// TwinCAT 3 PLC project PLC
// ProgramVersion: 3.1.4024.0
// libraries:
//   EfficientIO Communicator, * (EfficientIO)
//   EfficientIO Energy Basic, * (EfficientIO)
//   EfficientIO ModbusTCP, * (EfficientIO)
//   Lynus Energy ModbusRTU, * (Lynus AG)
//   Lynus Persistent Data V1, * (Lynus AG)
//   Lynus Standards, * (EfficientIO)
//   Tc2_Math, * (Beckhoff Automation GmbH)
//   Tc2_MBus, * (Beckhoff Automation GmbH)
//   Tc2_Standard, * (Beckhoff Automation GmbH)
//   Tc2_System, * (Beckhoff Automation GmbH)
//   Tc2_Utilities, * (Beckhoff Automation GmbH)
//   Tc3_JsonXml, * (Beckhoff Automation GmbH)
//   Tc3_Module, * (Beckhoff Automation GmbH)
// project tree:
//   / Fast_Task.TcTTO, Middle_Task.TcTTO, Slow_Task.TcTTO
//   FB/ FB_Delta_PV_Inverter_Sunspec.TcPOU (not stored), FB_KL6xxx_ModbusRTU_22B_Master.TcPOU, FB_Shelly_3EM.TcPOU (not stored), FB_Shelly_3EM_Helper.TcPOU (not stored), FB_Shelly_HT.TcPOU (not stored), FB_Shelly_HTplus.TcPOU (not stored), FB_Shelly_HTplus_Helper.TcPOU (not stored), FB_Shelly_HT_Helper.TcPOU
//   POUs/ MAIN.TcPOU, prgComEffIO.TcPOU (not stored), prgEM.TcPOU, prgEMS.TcPOU, prgGrid.TcPOU, prgHouse.TcPOU, prgMBUS.TcPOU, prgPersistent.TcPOU (not stored), prgPV.TcPOU, prgRWEffIO.TcPOU, prgVarEffIO.TcPOU (not stored)
// real-time tasks:
//   TASK Fast Task: cycle T#8ms, priority 8, ADS port 350
//   TASK Middle Task: cycle T#10ms, priority 10, ADS port 351
//   TASK Slow Task: cycle T#20ms, priority 20, ADS port 352
// I/O:
//   DEVICE Gerät 1 (Beckhoff CCAT)
//   DEVICE Gerät 2 (EtherCAT), AmsNetId 5.146.124.165.3.1
//     Klemme 1 (EK1200) [EK1200-5000 EtherCAT Netzteil (2A E-Bus)]
//       43A7_UV_Müller_Holzbau (EL3443-0010) [EL3443-0010 3K. Leistungsmessung 10A]
//       43A7.1_Abgang_Mieter (EL3443-0010) [EL3443-0010 3K. Leistungsmessung 10A]
//       43A8_Produktion_PV (EL3443-0010) [EL3443-0010 3K. Leistungsmessung 10A]
//       Klemme 5 (EL9010) [EL9010 Endklemme]
//   DEVICE Gerät 3 (RT-Ethernet Protocol), AmsNetId 5.146.124.165.4.1
//     BK9050 (BK9050-0000 192.168.1.118)
// variable links:
//   PLC/PLC Instance <-> Device 2 (EtherCAT)/Term 1 (EK1200)/43A7.1_Abgang_Mieter (EL3443-0010)
//     Middle_Task Inputs/prgHouse.ActivePowerTotal_2 <-> Total Active/Active Power
//   PLC/PLC Instance <-> Device 2 (EtherCAT)/Term 1 (EK1200)/43A7_UV_Müller_Holzbau (EL3443-0010)
//     Middle_Task Inputs/prgHouse.ActivePowerTotal_1 <-> Total Active/Active Power
//     Slow_Task Inputs/prgHouse.Strom1L1 <-> L1 Basic/Current
//     Slow_Task Inputs/prgHouse.Volt1L1 <-> L1 Basic/Voltage
//   PLC/PLC Instance <-> Device 2 (EtherCAT)/Term 1 (EK1200)/43A8_Produktion_PV (EL3443-0010)
//     Slow_Task Inputs/prgHouse.ActivePowerTotal_3 <-> Total Active/Active Power
//   PLC/PLC Instance <-> Device 3 (RT-Ethernet Protocol)/BK9050 (BK9050-0000 192.168.1.118)
//     Fast_Task Inputs/prgMBUS.stComIn @bit {16..184 step 8} <-> Term 2 (KL6781)/Channel 1/Data In {0..21}  (22 links)
//     Fast_Task Inputs/prgMBUS.stComIn <-> Term 2 (KL6781)/Channel 1/Status
//     Fast_Task Outputs/prgMBUS.stComOut <-> Term 2 (KL6781)/Channel 1/Ctrl
//     Fast_Task Outputs/prgMBUS.stComOut @bit {16..184 step 8} <-> Term 2 (KL6781)/Channel 1/Data Out {0..21}  (22 links)
//     Middle_Task Inputs/prgHouse.fbGrid1.fbKL3403.byStateCH1 <-> Elektromobilität (KL3403)/Channel 1/Status
//     Middle_Task Inputs/prgHouse.fbGrid1.fbKL3403.byStateCH2 <-> Elektromobilität (KL3403)/Channel 2/Status
//     Middle_Task Inputs/prgHouse.fbGrid1.fbKL3403.byStateCH3 <-> Elektromobilität (KL3403)/Channel 3/Status
//     Middle_Task Inputs/prgHouse.fbGrid1.fbKL3403.iDataInCH1 <-> Elektromobilität (KL3403)/Channel 1/Daten Ein
//     Middle_Task Inputs/prgHouse.fbGrid1.fbKL3403.iDataInCH2 <-> Elektromobilität (KL3403)/Channel 2/Daten Ein
//     Middle_Task Inputs/prgHouse.fbGrid1.fbKL3403.iDataInCH3 <-> Elektromobilität (KL3403)/Channel 3/Daten Ein
//     Middle_Task Inputs/prgHouse.fbGrid2.fbKL3403.byStateCH1 <-> Holzschnitzelheizung (KL3403)/Channel 1/Status
//     Middle_Task Inputs/prgHouse.fbGrid2.fbKL3403.byStateCH2 <-> Holzschnitzelheizung (KL3403)/Channel 2/Status
//     Middle_Task Inputs/prgHouse.fbGrid2.fbKL3403.byStateCH3 <-> Holzschnitzelheizung (KL3403)/Channel 3/Status
//     Middle_Task Inputs/prgHouse.fbGrid2.fbKL3403.iDataInCH1 <-> Holzschnitzelheizung (KL3403)/Channel 1/Daten Ein
//     Middle_Task Inputs/prgHouse.fbGrid2.fbKL3403.iDataInCH2 <-> Holzschnitzelheizung (KL3403)/Channel 2/Daten Ein
//     Middle_Task Inputs/prgHouse.fbGrid2.fbKL3403.iDataInCH3 <-> Holzschnitzelheizung (KL3403)/Channel 3/Daten Ein
//     Middle_Task Inputs/prgHouse.fbGrid3.fbKL3403.byStateCH1 <-> Lüftung_Kälte_Büro (KL3403)/Channel 1/Status
//     Middle_Task Inputs/prgHouse.fbGrid3.fbKL3403.byStateCH2 <-> Lüftung_Kälte_Büro (KL3403)/Channel 2/Status
//     Middle_Task Inputs/prgHouse.fbGrid3.fbKL3403.byStateCH3 <-> Lüftung_Kälte_Büro (KL3403)/Channel 3/Status
//     Middle_Task Inputs/prgHouse.fbGrid3.fbKL3403.iDataInCH1 <-> Lüftung_Kälte_Büro (KL3403)/Channel 1/Daten Ein
//     Middle_Task Inputs/prgHouse.fbGrid3.fbKL3403.iDataInCH2 <-> Lüftung_Kälte_Büro (KL3403)/Channel 2/Daten Ein
//     Middle_Task Inputs/prgHouse.fbGrid3.fbKL3403.iDataInCH3 <-> Lüftung_Kälte_Büro (KL3403)/Channel 3/Daten Ein
//     Middle_Task Outputs/prgHouse.fbGrid1.fbKL3403.byCntrCH1 <-> Elektromobilität (KL3403)/Channel 1/Kontrolle
//     Middle_Task Outputs/prgHouse.fbGrid1.fbKL3403.byCntrCH2 <-> Elektromobilität (KL3403)/Channel 2/Kontrolle
//     Middle_Task Outputs/prgHouse.fbGrid1.fbKL3403.byCntrCH3 <-> Elektromobilität (KL3403)/Channel 3/Kontrolle
//     Middle_Task Outputs/prgHouse.fbGrid2.fbKL3403.byCntrCH1 <-> Holzschnitzelheizung (KL3403)/Channel 1/Kontrolle
//     Middle_Task Outputs/prgHouse.fbGrid2.fbKL3403.byCntrCH2 <-> Holzschnitzelheizung (KL3403)/Channel 2/Kontrolle
//     Middle_Task Outputs/prgHouse.fbGrid2.fbKL3403.byCntrCH3 <-> Holzschnitzelheizung (KL3403)/Channel 3/Kontrolle
//     Middle_Task Outputs/prgHouse.fbGrid3.fbKL3403.byCntrCH1 <-> Lüftung_Kälte_Büro (KL3403)/Channel 1/Kontrolle
//     Middle_Task Outputs/prgHouse.fbGrid3.fbKL3403.byCntrCH2 <-> Lüftung_Kälte_Büro (KL3403)/Channel 2/Kontrolle
//     Middle_Task Outputs/prgHouse.fbGrid3.fbKL3403.byCntrCH3 <-> Lüftung_Kälte_Büro (KL3403)/Channel 3/Kontrolle

CONFIGURATION PLC
    RESOURCE PLC ON TwinCAT3
        TASK Fast_Task(INTERVAL := T#8ms, PRIORITY := 8);
        TASK Middle_Task(INTERVAL := T#10ms, PRIORITY := 10);
        TASK Slow_Task(INTERVAL := T#20ms, PRIORITY := 20);
        PROGRAM prgVarEffIO WITH Fast_Task : prgVarEffIO;
        PROGRAM prgRWEffIO WITH Fast_Task : prgRWEffIO;
        PROGRAM prgMBUS WITH Fast_Task : prgMBUS;
        PROGRAM prgPV WITH Fast_Task : prgPV;
        PROGRAM prgHouse WITH Middle_Task : prgHouse;
        PROGRAM prgGrid WITH Middle_Task : prgGrid;
        PROGRAM prgPersistent WITH Middle_Task : prgPersistent;
        PROGRAM prgEMS WITH Middle_Task : prgEMS;
        PROGRAM prgComEffIO WITH Slow_Task : prgComEffIO;
    END_RESOURCE
END_CONFIGURATION

// ---- POUs/prgRWEffIO.TcPOU
PROGRAM prgRWEffIO
VAR
	fbRW1		: FB_ReadWrite_V2;
END_VAR

fbRW1(
	eUploadType:= 3, // Change + 5 min Intervall 
	bBusy=> , 
	bError=> , 
	udiErrorCodeOut=> , 
	eErrorReadWrite_Out=> );

END_PROGRAM

// ---- POUs/prgMBUS.TcPOU
PROGRAM prgMBUS
VAR
	// M-Bus Kommunikation (KL6781)
	fbMBusKL6781         : FB_MBUSKL6781;             // Hauptbaustein für die M-Bus-Kommunikation
	stComIn              AT %I* : ST_KL6781inData22B; // Eingabestruktur für KL6781
	stComOut             AT %Q* : ST_KL6781outData22B;// Ausgabestruktur für KL6781
	stCom                : ST_MBUS_Communication;     // Kommunikationsstruktur für alle M-Bus-Geräte
	fbScann              : FB_MBUS_Scan;
	// Wärmezähler (Supercal 531)
	fbHolzkessel         : FB_MBUS_General;          	 // Funktionsbaustein für Holzkessel
	fbFussbodenheizung   : FB_MBUS_General;   		 	 // Funktionsbaustein für MAB Fußbodenheizung
	fbDSP_Produktion     : FB_MBUS_General;   			// Funktionsbaustein für DSP Produktion
	fbHeizkoerper_buero  : FB_MBUS_General;   			// Funktionsbaustein für Heizkörper Büro
	fbHalle_Bestand_S100 : FB_MBUS_General;   			// Funktionsbaustein für Halle Bestand S100
	fbLueftung	         : FB_MBUS_General;   			// Funktionsbaustein für Lüftung

	// Variablen für Steuerung
	m_Start1             : BOOL;                      
	m_Start2             : BOOL;                      
	m_Start3             : BOOL;
	m_Start4             : BOOL;
	m_Start5             : BOOL;
	m_Start6             : BOOL;
	
	//
	//TODO austausch FLOW mit Vorlauf und Rücklauftemperatur
	//
	
	// Ausgelesene Werte Wärmezähler
	lrEnergy_Holzkessel	 		: LREAL;								//{#lynus.ag#()}
	rFlow_Holzkessel     		: REAL;
	rPower_Holzkessel    		: REAL;									//{#lynus.ag#()}
	rflow_VL_Holzkessel			: REAL;									//{#lynus.ag#()}
	rflow_RL_Holzkessel			: REAL;									//{#lynus.ag#()}

	lrEnergy_Fussboden   		: LREAL;								//{#lynus.ag#()}
	rFlow_Fussboden         	: REAL;
	rPower_Fussboden        	: REAL;									//{#lynus.ag#()}
	rflow_VL_Fussboden			: REAL;									//{#lynus.ag#()}
	rflow_RL_Fussboden			: REAL;									//{#lynus.ag#()}

	lrEnergy_DSP_Produktion 	: LREAL;								//{#lynus.ag#()}
	rFlow_DSP_Produktion    	: REAL;
	rPower_DSP_Produktion   	: REAL;									//{#lynus.ag#()}
	rflow_VL_DSP_Produktion		: REAL;									//{#lynus.ag#()}
	rflow_RL_DSP_Produktion		: REAL;									//{#lynus.ag#()}
	
	lrEnergy_Heizkoerper_buero  : LREAL;								//{#lynus.ag#()}
	rFlow_Heizkoerper_buero     : REAL;
	rPower_Heizkoerper_buero    : REAL;									//{#lynus.ag#()}
	rflow_VL_Heizkoerper_buero	: REAL;									//{#lynus.ag#()}
	rflow_RL_Heizkoerper_buero	: REAL;									//{#lynus.ag#()}
	
	lrEnergy_Halle_Bestand_S100 : LREAL;								//{#lynus.ag#()}
	rFlow_Halle_Bestand_S100    : REAL;
	rPower_Halle_Bestand_S100   : REAL;									//{#lynus.ag#()}
	rflow_VL_Halle_Bestand_S100	: REAL;									//{#lynus.ag#()}
	rflow_RL_Halle_Bestand_S100	: REAL;									//{#lynus.ag#()}
	
	lrEnergy_Lueftung           : LREAL;								//{#lynus.ag#()}
	rFlow_Lueftung              : REAL;
	rPower_Lueftung             : REAL;									//{#lynus.ag#()}
	rflow_VL_Lueftung			: REAL;									//{#lynus.ag#()}
	rflow_RL_Lueftung			: REAL;									//{#lynus.ag#()}

	Err1 : E_MBUS_ERROR;
	Err2 : E_MBUS_ERROR;
	Err3 : E_MBUS_ERROR;
	Err4 : E_MBUS_ERROR;
	Err5 : E_MBUS_ERROR;
	Err6 : E_MBUS_ERROR;
	
	Busy1Trig : R_TRIG;
	DataReadyCount : DINT;
	DevError : ST_MBus_Info; 

	DataReadyCount2 : DINT;
	DevError2       : ST_MBus_Info; 

END_VAR

// ** M-Bus Hauptkommunikation **

fbMBusKL6781(
	usiRetries := 3,                    // Anzahl der Wiederholungen bei Fehler
	bStart := TRUE,                     // Startet die M-Bus-Kommunikation
	bDisabled := FALSE,                 // Deaktiviert die M-Bus-Kommunikation nicht
	bBusy => , 
	bReady => , 
	bError => , 
	eError => , 
	stComIn := stComIn, 
	stComOut := stComOut, 
	stCom := stCom
);

fbScann(
	bStart:= , 
	bStop:= , 
	eBaudrate:= E_MBUS_Baudrate.eMBus_Baud2400, 
	bDisabled:= , 
	bBusy=> , 
	bReady=> , 
	bError=> , 
	eError=> , 
	usiAddress=> , 
	usiCount=> , 
	arrDevice=> , 
	stCom:= stCom);


// ** Holzkessel (Supercal 531) auslesen **

//fbSupercal1.stSecAdr.udiIdNumber:= 30868639;

fbHolzkessel(
	usiAddress 	:= 1,                    	// M-Bus-Adresse(Primär)
	bStart 		:= m_Start1,                // Startflag
	usiUnit     := 1,               		// KW
	bDisabled 	:= FALSE,                 	
	bBusy => , 
	bReady => ,              				// Datenbereit-Status
	bError => , 
	eError => , 
	stCom 		:= stCom
);

IF NOT fbHolzkessel.bBusy AND fbHolzkessel.bError THEN

	Err1:= fbHolzkessel.eError;
END_IF

IF fbHolzkessel.bReady THEN

    lrEnergy_Holzkessel 	:= STRING_TO_REAL(fbHolzkessel.arrData[1].sValue);                 	// Energie (kWh)
    rFlow_Holzkessel 		:= STRING_TO_REAL(fbHolzkessel.arrData[6].sValue);                  // Durchfluss (m³/h)
    rPower_Holzkessel 	:= STRING_TO_REAL(fbHolzkessel.arrData[7].sValue);                    	// Leistung (kW)
END_IF

fbFussbodenheizung(
	usiAddress 	:= 2,                    	// M-Bus-Adresse(Primär)
	bStart 		:= m_Start2,                // Startflag
	usiUnit     := 1,               		// KW
	bDisabled 	:= FALSE,                 	
	bBusy => , 
	bReady => ,              				// Datenbereit-Status
	bError => , 
	eError => , 
	stCom 		:= stCom
);

IF NOT fbFussbodenheizung.bBusy AND fbFussbodenheizung.bError THEN

	Err2:= fbFussbodenheizung.eError;
END_IF

IF fbFussbodenheizung.bReady THEN

    lrEnergy_Fussboden 	:= STRING_TO_REAL(fbFussbodenheizung.arrData[1].sValue);                // Energie (kWh)
    rFlow_Fussboden 	:= STRING_TO_REAL(fbFussbodenheizung.arrData[6].sValue);                // Durchfluss (m³/h)
    rPower_Fussboden 	:= STRING_TO_REAL(fbFussbodenheizung.arrData[7].sValue);                // Leistung (kW)
	rflow_VL_Fussboden	:= STRING_TO_REAL(fbFussbodenheizung.arrData[3].sValue);					// Temperatur in Grad C
	rflow_RL_Fussboden	:= STRING_TO_REAL(fbFussbodenheizung.arrData[4].sValue);					// Temperatur in Grad C
END_IF

fbDSP_Produktion(
	usiAddress 	:= 3,                    	// M-Bus-Adresse(Primär)
	bStart 		:= m_Start3,                // Startflag
	usiUnit     := 1,               		// KW
	bDisabled 	:= FALSE,                 	
	bBusy => , 
	bReady => ,              				// Datenbereit-Status
	bError => , 
	eError => , 
	stCom 		:= stCom
);

IF NOT fbDSP_Produktion.bBusy AND fbDSP_Produktion.bError THEN

	Err3:= fbDSP_Produktion.eError;
END_IF

IF fbDSP_Produktion.bReady THEN

    lrEnergy_DSP_Produktion 	:= STRING_TO_REAL(fbDSP_Produktion.arrData[1].sValue);                 	// Energie (kWh)
    rFlow_DSP_Produktion 		:= STRING_TO_REAL(fbDSP_Produktion.arrData[6].sValue);                  // Durchfluss (m³/h)
    rPower_DSP_Produktion 		:= STRING_TO_REAL(fbDSP_Produktion.arrData[7].sValue);                  // Leistung (kW)
	rflow_VL_DSP_Produktion		:= STRING_TO_REAL(fbDSP_Produktion.arrData[3].sValue);					// Temperatur in Grad C
	rflow_RL_DSP_Produktion		:= STRING_TO_REAL(fbDSP_Produktion.arrData[4].sValue);					// Temperatur in Grad C
END_IF

fbHeizkoerper_buero(
	usiAddress 	:= 4,                    	// M-Bus-Adresse(Primär)
	bStart 		:= m_Start4,                // Startflag
	usiUnit     := 1,               		// KW
	bDisabled 	:= FALSE,                 	
	bBusy => , 
	bReady => ,              				// Datenbereit-Status
	bError => , 
	eError => , 
	stCom 		:= stCom
);

IF NOT fbHeizkoerper_buero.bBusy AND fbHeizkoerper_buero.bError THEN

	Err4:= fbHeizkoerper_buero.eError;
END_IF

IF fbHeizkoerper_buero.bReady THEN

    lrEnergy_Heizkoerper_buero 	:= STRING_TO_REAL(fbHeizkoerper_buero.arrData[1].sValue);                 	// Energie (kWh)
    rFlow_Heizkoerper_buero 	:= STRING_TO_REAL(fbHeizkoerper_buero.arrData[6].sValue);                  // Durchfluss (m³/h)
    rPower_Heizkoerper_buero 	:= STRING_TO_REAL(fbHeizkoerper_buero.arrData[7].sValue);                  // Leistung (kW)
	rflow_VL_Heizkoerper_buero	:= STRING_TO_REAL(fbHeizkoerper_buero.arrData[3].sValue);					// Temperatur in Grad C
	rflow_RL_Heizkoerper_buero	:= STRING_TO_REAL(fbHeizkoerper_buero.arrData[4].sValue);					// Temperatur in Grad C
END_IF

fbHalle_Bestand_S100(
	usiAddress 	:= 5,                    	// M-Bus-Adresse(Primär)
	bStart 		:= m_Start5,                // Startflag
	usiUnit     := 1,               		// KW
	bDisabled 	:= FALSE,                 	
	bBusy => , 
	bReady => ,              				// Datenbereit-Status
	bError => , 
	eError => , 
	stCom 		:= stCom
);

IF NOT fbHalle_Bestand_S100.bBusy AND fbHalle_Bestand_S100.bError THEN

	Err5:= fbHalle_Bestand_S100.eError;
END_IF

IF fbHalle_Bestand_S100.bReady THEN

    lrEnergy_Halle_Bestand_S100 	:= STRING_TO_REAL(fbHalle_Bestand_S100.arrData[1].sValue);                 	// Energie (kWh)
    rFlow_Halle_Bestand_S100 		:= STRING_TO_REAL(fbHalle_Bestand_S100.arrData[6].sValue);                  // Durchfluss (m³/h)
    rPower_Halle_Bestand_S100 		:= STRING_TO_REAL(fbHalle_Bestand_S100.arrData[7].sValue);                  // Leistung (kW)
	rflow_VL_Halle_Bestand_S100		:= STRING_TO_REAL(fbHalle_Bestand_S100.arrData[3].sValue);					// Temperatur in Grad C
	rflow_RL_Halle_Bestand_S100		:= STRING_TO_REAL(fbHalle_Bestand_S100.arrData[4].sValue);					// Temperatur in Grad C
END_IF


fbLueftung(
	usiAddress 	:= 6,                    	// M-Bus-Adresse(Primär)
	bStart 		:= m_Start6,                // Startflag
	usiUnit     := 1,               		// KW
	bDisabled 	:= FALSE,                 	
	bBusy => , 
	bReady => ,              				// Datenbereit-Status
	bError => , 
	eError => , 
	stCom 		:= stCom
);

IF NOT fbLueftung.bBusy AND fbLueftung.bError THEN

	Err6:= fbLueftung.eError;
END_IF

IF fbLueftung.bReady THEN

    lrEnergy_Lueftung 	:= STRING_TO_REAL(fbLueftung.arrData[1].sValue);             	// Energie (kWh)
    rFlow_Lueftung 		:= STRING_TO_REAL(fbLueftung.arrData[6].sValue);             	// Durchfluss (m³/h)
    rPower_Lueftung 	:= STRING_TO_REAL(fbLueftung.arrData[7].sValue);            	// Leistung (kW)
	rflow_VL_Lueftung	:= STRING_TO_REAL(fbLueftung.arrData[3].sValue);				// Temperatur in Grad C
	rflow_RL_Lueftung	:= STRING_TO_REAL(fbLueftung.arrData[4].sValue);				// Temperatur in Grad C
END_IF

END_PROGRAM

// ---- POUs/prgPV.TcPOU
PROGRAM prgPV
VAR
	//fbPV1							:FB_SunSpec_PV_Inverter;
	Wechselrichter1kWRaw AT %MW0	:INT;
	Wechselrichter1kW				:REAL;							//{#lynus.ag#()}
	Wechselrichter2kWRaw AT %MW2	:INT;
	Wechselrichter2kW				:REAL;							//{#lynus.ag#()}
	Wechselrichter3kWRaw AT %MW4	:INT;
	Wechselrichter3kW				:REAL;							//{#lynus.ag#()}
	Wechselrichter4kWRaw AT %MW6	:INT;
	Wechselrichter4kW				:REAL;							//{#lynus.ag#()}
	Wechselrichter5kWRaw AT %MW8	:INT;
	Wechselrichter5kW				:REAL;							//{#lynus.ag#()}
	Wechselrichter6kWRaw AT %MW10	:INT;
	Wechselrichter6kW				:REAL;							//{#lynus.ag#()}
	Wechselrichter7kWRaw AT %MW12	:INT;
	Wechselrichter7kW				:REAL;							//{#lynus.ag#()}
	Wechselrichter8kWRaw AT %MW14	:INT;
	Wechselrichter8kW				:REAL;							//{#lynus.ag#()}
	Wechselrichter9kWRaw AT %MW16	:INT;
	Wechselrichter9kW				:REAL;							//{#lynus.ag#()}
	PV_Gesamt						:REAL;							//{#lynus.ag#()}

END_VAR

Wechselrichter1kW := TO_REAL(Wechselrichter1kWRaw) / 100.0;
Wechselrichter2kW := TO_REAL(Wechselrichter2kWRaw) / 100.0;
Wechselrichter3kW := TO_REAL(Wechselrichter3kWRaw) / 100.0;
Wechselrichter4kW := TO_REAL(Wechselrichter4kWRaw) / 100.0;
Wechselrichter5kW := TO_REAL(Wechselrichter5kWRaw) / 100.0;
Wechselrichter6kW := TO_REAL(Wechselrichter6kWRaw) / 100.0;
Wechselrichter7kW := TO_REAL(Wechselrichter7kWRaw) / 100.0;
Wechselrichter8kW := TO_REAL(Wechselrichter8kWRaw) / 100.0;
Wechselrichter9kW := TO_REAL(Wechselrichter9kWRaw) / 100.0;

PV_Gesamt 		  := Wechselrichter1kW + Wechselrichter2kW + Wechselrichter3kW + Wechselrichter4kW + Wechselrichter5kW + Wechselrichter6kW + Wechselrichter7kW + Wechselrichter8kW + Wechselrichter9kW;

(*
fbPV1(
	bEnable:= , 
	sIPAdress:= '192.168.140.6', 
	byUnitID_Inverter:= 1, 
	stDataSunSpec=> , 
	stDataEMPower_PV=> , 
	stDataEMCounter_PV=> , 
	diNrOfEM_OUT_PV=> 
);
*)

END_PROGRAM

// ---- POUs/prgHouse.TcPOU
PROGRAM prgHouse
VAR
	fbKBusState					: FB_K_Bus_State;
	uint_KBusState				: UINT;							//{#lynus.ag#()}
	lrHousePower				: LREAL;								//{#lynus.ag#()}
	lrNetzEinspeisung			: LREAL;								//{#lynus.ag#()}
	lrBetriebMuellerBau			: LREAL;								//{#lynus.ag#()}
	lrElektromobilitaet			: LREAL;								//{#lynus.ag#()}
	lrHolzschnitzel				: LREAL;								//{#lynus.ag#()}
	lrLueftung_Kaelte			: LREAL;								//{#lynus.ag#()}
	//rPVProd						: REAL;									//{#lynus.ag#()}
	lrAbgaenge					: REAL;									//{#lynus.ag#()}
	fbGrid1						: FB_EM_Beckhoff_KL3403;  	//Elektromobilität 
	fbGrid2						: FB_EM_Beckhoff_KL3403;	//Holzschnitzelheizung
	fbGrid3						: FB_EM_Beckhoff_KL3403;	//Lüftung/Kälte Büro
	
	

    Volt1L1  AT %I* : REAL;
    Strom1L1 AT %I* : REAL;
	//UV Müller Holzbau
	ActivePowerTotal_1	AT %I*	: REAL;									//{#lynus.ag#()}
	//Abgang Direktmessung
	ActivePowerTotal_2	AT %I*	: REAL;									//{#lynus.ag#()}
	//Produktion PV
	ActivePowerTotal_3	AT %I*	: REAL;									//{#lynus.ag#()}

END_VAR

lrNetzEinspeisung := ActivePowerTotal_1/1000 + ActivePowerTotal_2/1000 - prgPV.PV_Gesamt;

lrElektromobilitaet	:= fbGrid1.stDataEMPower.lrPowerTotal;
lrHolzschnitzel		:= fbGrid2.stDataEMPower.lrPowerTotal;
lrLueftung_Kaelte	:= fbGrid3.stDataEMPower.lrPowerTotal;
lrHousePower		:= ActivePowerTotal_1/1000 + fbGrid1.stDataEMPower.lrPowerTotal + fbGrid2.stDataEMPower.lrPowerTotal + fbGrid3.stDataEMPower.lrPowerTotal;

lrBetriebMuellerBau := -fbGrid1.stDataEMPower.lrPowerTotal - fbGrid2.stDataEMPower.lrPowerTotal - fbGrid3.stDataEMPower.lrPowerTotal + lrHousePower;	

//rPVProd				:= (ActivePowerTotal_3)/100 * -1;					//Invertieren
lrAbgaenge 			:= ActivePowerTotal_2/1000;
//lrHousePower 		:= lrBetriebMuellerBau * -1;						//Invertierte Einspeisung für Darstellung

//The mapping of this function must be linked with the K-Bus State in the E/A Part
fbKBusState(	uiKBusState_OUT=> , 
				b_Kbus_notOk=> , 
				word_ErrorCount=> );

fbGrid1(
	bEnable:= TRUE, 
	bChannel1Invers:= FALSE, 
	bChannel2Invers:= FALSE, 
	bChannel3Invers:= FALSE, 
	uiCurrentTransformerRatioL1:= 400, 
	uiCurrentTransformerRatioL2:= 400, 
	uiCurrentTransformerRatioL3:= 400, 
	uiKBusState_IN:= fbKBusState.uiKBusState_OUT, 
	stDataEMPower=> , 
	stDataEMCounter=> , 
	stDataEMPowerRealTime=> , 
	stDataEMCounterRealTime=> , 
	diNrOfEM_OUT=> );
	
	
fbGrid2(
	bEnable:= TRUE, 
	bChannel1Invers:= FALSE, 
	bChannel2Invers:= FALSE, 
	bChannel3Invers:= FALSE, 
	uiCurrentTransformerRatioL1:= 400, 
	uiCurrentTransformerRatioL2:= 400, 
	uiCurrentTransformerRatioL3:= 400, 
	uiKBusState_IN:= , 
	stDataEMPower=> , 
	stDataEMCounter=> , 
	stDataEMPowerRealTime=> , 
	stDataEMCounterRealTime=> , 
	diNrOfEM_OUT=> );
	
fbGrid3(
	bEnable:= TRUE, 
	bChannel1Invers:= FALSE, 
	bChannel2Invers:= FALSE, 
	bChannel3Invers:= FALSE, 
	uiCurrentTransformerRatioL1:= 400, 
	uiCurrentTransformerRatioL2:= 400, 
	uiCurrentTransformerRatioL3:= 400, 
	uiKBusState_IN:= , 
	stDataEMPower=> , 
	stDataEMCounter=> , 
	stDataEMPowerRealTime=> , 
	stDataEMCounterRealTime=> , 
	diNrOfEM_OUT=> );

END_PROGRAM

// ---- POUs/prgGrid.TcPOU
PROGRAM prgGrid
VAR
	fbKBusState					: FB_K_Bus_State;
	fbGrid						: FB_EM_Beckhoff_KL3403;
	uint_KBusState				: UINT;							//{#lynus.ag#()}
	fbGridCounter				: FB_EnergyCounter;
	lrGridPower					: LREAL;								//{#lynus.ag#()}
	lrVoltage_L1N					: LREAL;								//{#lynus.ag#()}
	lrVoltage_L2N					: LREAL;								//{#lynus.ag#()}
	lrVoltage_L3N					: LREAL;								//{#lynus.ag#()}
END_VAR
VAR PERSISTENT
	rSizeGridConn				: REAL;									//{#lynus.ag#()}
	lrCounterGridProd			: LREAL;								//{#lynus.ag#()}
	lrCounterGridCons			: LREAL;								//{#lynus.ag#()}
END_VAR

//The mapping of this function must be linked with the K-Bus State in the E/A Part
fbKBusState(	uiKBusState_OUT=> , 
				b_Kbus_notOk=> , 
				word_ErrorCount=> );

//The mapping of this function must be linked with the KL3403 in the E/A Part
//UV1
fbGrid(
	bEnable:= TRUE, 
	bChannel1Invers:= FALSE,				//Invert power data when transformer are mounted upside down
	bChannel2Invers:= FALSE,			// CT seems to be wired the wrong wy around
	bChannel3Invers:= FALSE,
	uiCurrentTransformerRatioL1:= 400, //Transformer ratio on the secondary side
	uiCurrentTransformerRatioL2:= 400, 
	uiCurrentTransformerRatioL3:= 400, 
	uiKBusState_IN:= fbKBusState.uiKBusState_OUT, 
	stDataEMPower=> , 
	stDataEMCounter=> , 
	stDataEMPowerRealTime=> , 
	stDataEMCounterRealTime=> , 
	diNrOfEM_OUT=> );
	
uint_KBusState :=	fbKBusState.uiKBusState_OUT;
lrGridPower := fbGrid.stDataEMPower.lrPowerTotal;

// EnergyCounter
fbGridCounter(
	byActiveTariff:= 1, 
	lrPowerInput:= lrGridPower, 
	lrTotalCounterEnergy_Consumption=> , 
	lrTotalCounterEnergy_Production=> , 
	lrCounterEnergyT1_Consumption=> , 
	lrCounterEnergyT2_Consumption=> , 
	lrCounterEnergyT1_Production=> , 
	lrCounterEnergyT2_Production=> );

IF fbGridCounter.lrTotalCounterEnergy_Production > lrCounterGridProd THEN  	
		lrCounterGridProd := fbGridCounter.lrTotalCounterEnergy_Production;
END_IF

IF fbGridCounter.lrTotalCounterEnergy_Consumption > lrCounterGridCons THEN  	
	lrCounterGridCons := fbGridCounter.lrTotalCounterEnergy_Consumption;
END_IF

lrVoltage_L1N := fbGrid.stDataEMPower.lrVoltageL1N;
lrVoltage_L2N := fbGrid.stDataEMPower.lrVoltageL2N;
lrVoltage_L3N := fbGrid.stDataEMPower.lrVoltageL3N;

END_PROGRAM

// ---- POUs/prgEMS.TcPOU
PROGRAM prgEMS
VAR PERSISTENT
	byMaxDepthOfDischrgEPO		: BYTE;							//{#lynus.ag#()}
	byPrioMinChrgBattSOCInEPO	: BYTE;							//{#lynus.ag#()}
	byResChrgfromGridToBatt		: BYTE;							//{#lynus.ag#()}
	byReserveSOCEPO				: BYTE;							//{#lynus.ag#()}
	uiUpdateTime				: UINT;							//{#lynus.ag#()}
	bEnableEMS					: BOOL;							//{#lynus.ag#()}
	bAllowChrgFromGrid			: BOOL;							//{#lynus.ag#()}
	rMainFuseCSEMS				: REAL;							//{#lynus.ag#()}
	iOperationModeEMS			: INT;							//{#lynus.ag#()}
	rSizeGridConn				: REAL;							//{#lynus.ag#()}
END_VAR
VAR
	fbEMS						: FB_EMS_V2;
	bIsEnableEMS				: BOOL;							//{#lynus.ag#()}
	bStateAllowChrgFromGrid		: BOOL;							//{#lynus.ag#()}
	bStateFuseCS				: BOOL;							//{#lynus.ag#()}
	bHPActivate					: BOOL;							//{#lynus.ag#()}
	bControllingState			: BOOL;							//{#lynus.ag#()}
	iMessageEMS					: INT;							//{#lynus.ag#()}
	rHeartbeatEMS				: REAL;							//{#lynus.ag#()}
	rErrorWarningEMS			: REAL;							//{#lynus.ag#()}
	rReadyEMS					: REAL;							//{#lynus.ag#()}
	rNewBatteryPowerEMS			: REAL;							//{#lynus.ag#()}
	fbGrid: FB_Grid_Power_Ext_Input;

END_VAR

IF iOperationModeEMS = 0 THEN fbEMS.eOperationMode := E_OperatingMode_EMS.eAllOff;
ELSIF iOperationModeEMS = 1 THEN fbEMS.eOperationMode := E_OperatingMode_EMS.eSelfConsumption;	
ELSIF iOperationModeEMS = 2 THEN fbEMS.eOperationMode := E_OperatingMode_EMS.ePeakLoadCapping;
ELSIF iOperationModeEMS = 3 THEN fbEMS.eOperationMode := E_OperatingMode_EMS.eLoadManagement;			
END_IF
fbEMS.stSetupEMS.bAllowChrgFromGrid := bAllowChrgFromGrid;
fbEMS.stSetupEMS.byMaxDepthOfDischrgEPO := byMaxDepthOfDischrgEPO;
// fbEMS.stSetupEMS.byPrioMinChrgBattSOCInEPO := byPrioMinChrgBattSOCInEPO;
// fbEMS.stSetupEMS.byResChrgfromGridToBatt := byResChrgfromGridToBatt;
fbEMS.stSetupEMS.byReserveSOCEPO := byReserveSOCEPO;
//fbEMS.stSetupEMS.rSizeMainFuseCS := rMainFuseCSEMS;
fbEMS.stSizeMainFuseCS.rElSizeLine1 := rMainFuseCSEMS;
fbEMS.stSetupEMS.bEnableMainFuseFunc := bStateFuseCS;
fbEMS.stSetupEMS.uiUpdateTime := uiUpdateTime;

fbEMS(
	bEnable						:= bEnableEMS, 
//	diNrOfEM_IN_ECS				:= , 
	stSetupEMS					:= , 
	eOperationMode				:= , 
	eSpeedModeBackendController	:= E_SpeedModeBackendController_EMS.eFast, 
	eSpeedModeLocalController	:= E_SpeedModeLocalController_EMS.eFast,
	bActivateHP					:= bHPActivate, 
	bControllingState			:= bControllingState, 
	rHeartbeat					:= rHeartbeatEMS, 
	rErrorWarning				:= rErrorWarningEMS, 
	rEnergyOptReady				:= rReadyEMS, 
	rNewBattPower				:= rNewBatteryPowerEMS, 

	eMessageEMS				=> iMessageEMS, 
	bStateEnable			=> bIsEnableEMS, 
	bStateAllowChrgFromGrid	=> bStateAllowChrgFromGrid, 
	bMissingPowerData		=> , 
	bSurplusAvailable		=> , 
	byProgress				=> , 
	uiState_OUT				=> , 
	diNrOfEMS_OUT			=> , 
	arrMinPrioReached		=> , 
	arrMaxPrioReached		=> ,
	);
	
fbGrid(
	bEnable:= TRUE, 
	diNrOfEMS_IN:= prgEMS.fbEMS.diNrOfEMS_OUT, 
	rSizeGridConn:= rSizeGridConn , 
	bExtErrorGrid:= , 
	lrExtGridPower:= prgHouse.lrNetzEinspeisung , 
	lrExtTotalCounterEnergy_Consumption:= , 
	lrExtTotalCounterEnergy_Production:= , 
	lrExtCounterEnergyT1_Consumption:= , 
	lrExtCounterEnergyT2_Consumption:= , 
	lrExtCounterEnergyT1_Production:= , 
	lrExtCounterEnergyT2_Production:= , 
	stDataGrid=> , 
	diNrOfGrid_OUT=> );

END_PROGRAM

// ---- FB/FB_KL6xxx_ModbusRTU_22B_Master.TcPOU
FUNCTION_BLOCK FB_KL6xxx_ModbusRTU_22B_Master
VAR_INPUT
	bConfigTerminal							: BOOL;																		//Possibility to configure the Terminal manually (Its only possible when the Terminal is not configured successfully)
	uiKBusState_IN							: UINT;																		//K-Bus State from the K-Bus Box on wich the Terminal is connected. (Connect with FB_K_Bus_state)
END_VAR
VAR_OUTPUT
	bBusy									: BOOL;																		//Function is Busy
	byErrorWarning							: BYTE;																		//Error Warning State
	byActualAdressInUse						: BYTE;																		//Actual Modbus Adress in Use
	diNrOfMBRTUMasterLine_OUT				: DINT;																		//Active Number from the RTU Master Function for using on other functions
	eMessageMBRTUMaster						: E_Message_MBRTUMaster;													//Message from the RTU Master Function
END_VAR				
VAR_OUTPUT PERSISTENT
	bTerminalIsConfigured					: BOOL;																		//Its True when the configuration is successfully
END_VAR
VAR		
	config_execute							: BOOL ;
	//{attribute 'hide'}
	fbKL6xxxConfig							: KL6configuration;															//FB KL6xxx to config the terminal
	fbmodbusmaster							: ModbusRtuMaster_KL6x22B;													//FB Modbus RTU
	{attribute 'hide'}
	fbmodbusmaster_Init						: ModbusRtuMaster_KL6x22B;													//FB Modbus RTU Master for workaroud regarding the internal Beckhoff problem in this function
	{attribute 'hide'}
	fbNumberDevice							: FB_NumberOfDevice;														//Function block to calcualte the number of the Device	
	{attribute 'hide'}
	fbModbusRTUMessage						: FB_MBRTUMaster_Messages;													//Modbus RTU Messages	
	{attribute 'hide'}
	FPConfigManual							: R_TRIG;																	//Internal positive Edge
	{attribute 'hide'}
	FPConfigAuto							: R_TRIG;																	//Internal positive Edge
	{attribute 'hide'}
	FPProcessCompleted						: R_TRIG;																	//Internal positive Edge
	{attribute 'hide'}
	FPError									: R_TRIG;																	//Internal positive Edge
	{attribute 'hide'}
	FPErrorIsActive							: R_TRIG;																	//Internal positive Edge
	{attribute 'hide'}
	FNInitSmall								: F_TRIG;																	//Internal negative Edge
	{attribute 'hide'}
	FNBusy									: F_TRIG;																	//Internal negative Edge
	{attribute 'hide'}
	timInit									: TON;																		//Delay to start the Terminal Configuration after the start from the plc
	{attribute 'hide'}
	timTimout								: TON;																		//Timer Timout to go on next Modbus Adress when the Ack is not set back to False
	{attribute 'hide'}
	timDissableFunctions					: TON;																		//Timer to dissable the Function after Lynus_Standards.Constants_General.tTimeDissableLynusFunctions Days without connection to the Lynus Cloud
	{attribute 'hide'}
	timResetConnectionOnGVL					: TON;																		//Timer to try reset the connection Flag on the GVL. (When somebody delete the Connection Function and make only a onlinechange)
	{attribute 'hide'}
	arrPD									: ARRAY[1..2] OF FB_PersistentData_Number;									//Function to save persistent data
	{attribute 'hide'}
	bTakeActualAdress						: BOOL;																		//True if the Current address is to be used
	{attribute 'hide'}
	bAdressHasChanged						: BOOL;																		//True if the Adress has changed
	{attribute 'hide'}
	bErrorIsActive							: BOOL;																		//True if a Error is happend. False after the next successfully read or write command
	{attribute 'hide'}
	bStopReadWrite							: BOOL;																		//Stop Function because Modbus Adress has chaged
	{attribute 'hide'}
	byLPSmallestAdress						: BYTE;																		//Loop to find out the smallest Modbus Adress
	{attribute 'hide'}
	byLPBiggestAdress						: BYTE;																		//Loop to find out the biggest Modbus Adress
	{attribute 'hide'}
	byLPActualAdress						: BYTE;																		//Loop to find out the next actuall adress
	{attribute 'hide'}
	byLPNumbersOfTotalSlaves				: BYTE;																		//Loop to find out the number of total Modbus Slaves
	{attribute 'hide'}
	bySmallestAdress						: BYTE;																		//Smallest Modbus Adress
	{attribute 'hide'}
	byBiggestAdress							: BYTE;																		//Biggest Modbus Adress
	{attribute 'hide'}
	byActualAdressInUse_CP					: BYTE;																		//Actual Modbus Adress in Use to compare it with the old one
	{attribute 'hide'}
	byNumberOfTotalSlaves					: BYTE;																		//Number of all Modbus Slaves
	{attribute 'hide'}
	byWaitInStep							: BYTE;																		//Wait in Step before start to clean data on PLC
	{attribute 'hide'}
	byLPMBAdress							: BYTE;																		//Loop for manage new Modbus Adress List after a change
	{attribute 'hide'}
	bySearchMBAdress						: BYTE;																		//Search Modbus Adress after change
	{attribute 'hide'}
	byPosInArrayMBAdress					: BYTE;																		//Save new Range from Modbus adress in the Array after a change
	{attribute 'hide'}
	iStateGVLData							: INT;																		//State machine to handle the data on the GVL
	{attribute 'hide'}
	iStateSetMBAdress						: INT;																		//State machin eto order the Modbus Adress after a change
	{attribute 'hide'}
	diCounterForGVL							: DINT;																		//Counter to clean old data on GVL
	{attribute 'hide'}
	arrRead									: ARRAY[1..Constants_Bussystems.wQuantityOfRegistersMBRTUMaster] OF WORD;	//Puffer for read out data
	{attribute 'hide'}
	arrMBAdress								: ARRAY[1..247] OF BYTE;													//Array with the actual Modbus Adress Config
END_VAR
VAR PERSISTENT
	{attribute 'conditionalshow'}
	eDeviceType								: E_MBRTUMaster_DeviceType;													//Device Type on witch the Terminal is configured
END_VAR

//Creator : Kai Ebensperger
//Company : Lynus AG
//Date : 08.07.2021
//Version : 1.0.0.0

//With this FB a serial 22 byte terminal can be configured and data can be sent/received via Modbus RTU.
//Only devices of the same type may be operated on the same master (because its not good to write to much new configurations on the terminal).
//The 1 slave that is called before the master FB in the PLC code configures the terminal
//The block must be called in a task of 5MS
//The system works according to the Master Slave principle
//Multiple communication is not possible in RTU principle

//NOTE for diNr.....Designation => 
//_IN = Here Data come in from other Functions or go out to other functions about the GVL
//_OUT = Here Data go out to other functions about the GVL

(*-------------------------------------------------------------Calcualte the number of RTU Master---------------------------------------------------------------*)

fbNumberDevice(
	diActualNumberOfDevices:= Lynus_Standards.GVL_Bussystems.diNumberOfMBRTUMasters, 
	diMaxNumberOfDevices:= Constants_Bussystems.diMaxNumberOfMBRTUMasterKL6xxx, 
	udiCounterOnlineChange:= TwinCAT_SystemInfoVarList._AppInfo.OnlineChangeCnt, 
	bNumberIsCalculatet=> , 
	bFPNumberIsCalculatet=> , 
	bOnlineChange=> , 
	diNumberForThisDevice=> diNrOfMBRTUMasterLine_OUT, 
	diNumberOfTotalDevices=> );

//Write new Numer on GVL
IF fbNumberDevice.bFPNumberIsCalculatet THEN
	Lynus_Standards.GVL_Bussystems.diNumberOfMBRTUMasters := fbNumberDevice.diNumberOfTotalDevices;	
END_IF 

//Delete old Number on GVL
IF fbNumberDevice.bOnlineChange THEN 
	Lynus_Standards.GVL_Bussystems.diNumberOfMBRTUMasters := diNrOfMBRTUMasterLine_OUT;	
		iStateGVLData := 1; 
END_IF	
	
(*-------------------------------------------------------------Service from Backend is ready and check the connection to backen for dissabel/enable Function---------------------------------------------------------------*)

//Try to reset the variable for connection on the GVL. When all is normal then the Lynus Mqtt connection function set this variable to true in the next cycle
//When we have no connection to the backend then after Lynus_Standards.Constants_General.tTimeDissableLynusFunctions days the Function is dissabled with all of his functionalities
timResetConnectionOnGVL(IN:= NOT timResetConnectionOnGVL.Q, PT:= T#1H, Q=> , ET=> );
	IF timResetConnectionOnGVL.Q THEN Lynus_Standards.GVL_Communicator.bStateConnectionToEnableFunctions := FALSE; END_IF
		IF NOT Lynus_Standards.GVL_Communicator.bStateConnectionToEnableFunctions THEN timDissableFunctions.IN := TRUE; ELSE timDissableFunctions.IN := FALSE; END_IF  
			timDissableFunctions(IN:= , PT:= Lynus_Standards.Constants_General.tTimeDissableLynusFunctions, Q=> , ET=> );

(*------------------------------------------------------------------Configuration----------------------------------------------------------------------------*)
			
//Configurate the seriall Terminal
//The configuration is depending what Slave is connected to the terminal
timInit(IN:= Lynus_Standards.GVL_Bussystems.stDataOfMBRTUMasterKL6xxx[diNrOfMBRTUMasterLine_OUT].eMBRTUDeviceType <> E_MBRTUMaster_DeviceType.eNoModbusRTUDevice AND uiKBusState_IN = 0, PT:=T#500MS, Q=> , ET=> );

IF Lynus_Standards.GVL_Bussystems.stDataOfMBRTUMasterKL6xxx[diNrOfMBRTUMasterLine_OUT].eMBRTUDeviceType <> eDeviceType AND timInit.Q THEN
	FPConfigAuto.CLK := TRUE;
		eDeviceType := Lynus_Standards.GVL_Bussystems.stDataOfMBRTUMasterKL6xxx[diNrOfMBRTUMasterLine_OUT].eMBRTUDeviceType;
ELSE
	FPConfigAuto.CLK := FALSE;
END_IF 	 

FPConfigAuto(CLK:= , Q=> );

//Configuration from the Terminal by the Slave Type
IF Lynus_Standards.GVL_Bussystems.stDataOfMBRTUMasterKL6xxx[diNrOfMBRTUMasterLine_OUT].eMBRTUDeviceType = E_MBRTUMaster_DeviceType.ePilotPMAC201_HW THEN
	//Pilot PMAC201 HW Energymessurement Device
	fbKL6xxxConfig.Mode := SERIALLINEMODE_KL6_22B_STANDARD;
	fbKL6xxxConfig.Baudrate := 38400;
	fbKL6xxxConfig.NoDatabits := 8;
	fbKL6xxxConfig.Parity := PARITY_NONE;
	fbKL6xxxConfig.Stopbits := 1;
	fbKL6xxxConfig.Handshake := RS485_HALFDUPLEX;
	fbKL6xxxConfig.ContinousMode := FALSE;
	//Timout	
	timTimout.PT := T#2S;
	fbmodbusmaster.Timeout := T#2S;
ELSIF Lynus_Standards.GVL_Bussystems.stDataOfMBRTUMasterKL6xxx[diNrOfMBRTUMasterLine_OUT].eMBRTUDeviceType = E_MBRTUMaster_DeviceType.eDrexelAWeiss_AereosilentStratosLU_Ventilation THEN
	//Aereosilent Stratos Ventilation Drexel and Weiss
	fbKL6xxxConfig.Mode := SERIALLINEMODE_KL6_22B_STANDARD;
	fbKL6xxxConfig.Baudrate := 19200;
	fbKL6xxxConfig.NoDatabits := 8;
	fbKL6xxxConfig.Parity := PARITY_NONE;
	fbKL6xxxConfig.Stopbits := 1;
	fbKL6xxxConfig.Handshake := HANDSHAKE_NONE;
	fbKL6xxxConfig.ContinousMode := FALSE;
	//Timout	
	timTimout.PT := T#10S;
	fbmodbusmaster.Timeout := T#3S;
ELSIF Lynus_Standards.GVL_Bussystems.stDataOfMBRTUMasterKL6xxx[diNrOfMBRTUMasterLine_OUT].eMBRTUDeviceType = E_MBRTUMaster_DeviceType.eABB_CM_UFD_M31M_NAProtection THEN
	//CM_UFD_M31M ABB NA Protection
	fbKL6xxxConfig.Mode := SERIALLINEMODE_KL6_22B_STANDARD;
	fbKL6xxxConfig.Baudrate := 38400;
	fbKL6xxxConfig.NoDatabits := 8;
	fbKL6xxxConfig.Parity := PARITY_NONE;
	fbKL6xxxConfig.Stopbits := 1;
	fbKL6xxxConfig.Handshake := RS485_HALFDUPLEX;
	fbKL6xxxConfig.ContinousMode := FALSE;
	//Timout	
	timTimout.PT := T#2S;
	fbmodbusmaster.Timeout := T#1S;
ELSIF Lynus_Standards.GVL_Bussystems.stDataOfMBRTUMasterKL6xxx[diNrOfMBRTUMasterLine_OUT].eMBRTUDeviceType = E_MBRTUMaster_DeviceType.eSchrack_ECS_CIONHOME_SEMIPUBLIC THEN
	//Schrack Electric Charging Station CionHome and Semipublic
	fbKL6xxxConfig.Mode := SERIALLINEMODE_KL6_22B_STANDARD;
	fbKL6xxxConfig.Baudrate := 57600;
	fbKL6xxxConfig.NoDatabits := 8;
	fbKL6xxxConfig.Parity := PARITY_NONE;
	fbKL6xxxConfig.Stopbits := 1;
	fbKL6xxxConfig.Handshake := RS485_HALFDUPLEX;
	fbKL6xxxConfig.ContinousMode := FALSE;
	//Timout	
	timTimout.PT := T#2S;
	fbmodbusmaster.Timeout := T#2S;
ELSIF Lynus_Standards.GVL_Bussystems.stDataOfMBRTUMasterKL6xxx[diNrOfMBRTUMasterLine_OUT].eMBRTUDeviceType = E_MBRTUMaster_DeviceType.ePV_DeltaSunspec THEN
	//Delte PV Inverter with Sunspec Protocol
	fbKL6xxxConfig.Mode := SERIALLINEMODE_KL6_22B_STANDARD;
	fbKL6xxxConfig.Baudrate := 19200;
	fbKL6xxxConfig.NoDatabits := 8;
	fbKL6xxxConfig.Parity := PARITY_NONE;
	fbKL6xxxConfig.Stopbits := 1;
	fbKL6xxxConfig.Handshake := RS485_HALFDUPLEX;
	fbKL6xxxConfig.ContinousMode := FALSE;
	//Timout	
	timTimout.PT := T#2S;
	fbmodbusmaster.Timeout := T#2S;
END_IF

FPConfigManual(CLK:= bConfigTerminal, Q=> );

fbKL6xxxConfig(
//	Execute := config_execute,
	Execute:= (FPConfigAuto.Q AND NOT bTerminalIsConfigured) OR (timInit.Q AND NOT bTerminalIsConfigured AND FPConfigManual.Q), 
	Mode:= ,
	Baudrate:= , 
	NoDatabits:= , 
	Parity:= , 
	Stopbits:= , 
	Handshake:= , 
	ContinousMode:= , 
	pComIn:= ADR(fbmodbusmaster.InData), 
	pComOut:= ADR(fbmodbusmaster.OutData), 
	SizeComIn:= SIZEOF(fbmodbusmaster.InData),
	Done=> , 
	Busy=> , 
	Error=> , 
	ErrorId=> );

IF fbKL6xxxConfig.Done THEN
	bTerminalIsConfigured := TRUE;

ELSIF NOT fbKL6xxxConfig.Busy AND fbKL6xxxConfig.Error THEN
	// ToDo bei Fehler neu anstossen.
	//
END_IF

(*------------------------------------------------------------------Read-Write----------------------------------------------------------------------------*)
	 
//Choose the right Modbus RTU Action for Read or Write Data
IF Lynus_Standards.GVL_Bussystems.stDataOfMBRTUMasterKL6xxx[diNrOfMBRTUMasterLine_OUT].eMBRTUReadWriteMode = E_MBRTUMaster_ReadWriteMode.eModbusRTUMaster_Diagnostics THEN 
	fbmodbusmaster.Diagnostics(); 
		fbmodbusmaster.cbLength := SIZEOF(Lynus_Standards.GVL_Bussystems.stDataOfMBRTUMasterKL6xxx[diNrOfMBRTUMasterLine_OUT].arrWriteOutData);
			fbmodbusmaster.pMemoryAddr := ADR(Lynus_Standards.GVL_Bussystems.stDataOfMBRTUMasterKL6xxx[diNrOfMBRTUMasterLine_OUT].arrWriteOutData);
END_IF
IF Lynus_Standards.GVL_Bussystems.stDataOfMBRTUMasterKL6xxx[diNrOfMBRTUMasterLine_OUT].eMBRTUReadWriteMode = E_MBRTUMaster_ReadWriteMode.eModbusRTUMaster_ReadCoils THEN 
	fbmodbusmaster.ReadCoils(); 
		fbmodbusmaster.cbLength := SIZEOF(arrRead);
			fbmodbusmaster.pMemoryAddr := ADR(arrRead);	
END_IF
IF Lynus_Standards.GVL_Bussystems.stDataOfMBRTUMasterKL6xxx[diNrOfMBRTUMasterLine_OUT].eMBRTUReadWriteMode = E_MBRTUMaster_ReadWriteMode.eModbusRTUMaster_ReadInputRegs THEN 
	fbmodbusmaster.ReadInputRegs(); 
		fbmodbusmaster.cbLength := SIZEOF(arrRead);
			fbmodbusmaster.pMemoryAddr := ADR(arrRead);
END_IF
IF Lynus_Standards.GVL_Bussystems.stDataOfMBRTUMasterKL6xxx[diNrOfMBRTUMasterLine_OUT].eMBRTUReadWriteMode = E_MBRTUMaster_ReadWriteMode.eModbusRTUMaster_ReadInputStatus THEN 
	fbmodbusmaster.ReadInputStatus(); 
		fbmodbusmaster.cbLength := SIZEOF(arrRead);
			fbmodbusmaster.pMemoryAddr := ADR(arrRead);
END_IF
IF Lynus_Standards.GVL_Bussystems.stDataOfMBRTUMasterKL6xxx[diNrOfMBRTUMasterLine_OUT].eMBRTUReadWriteMode = E_MBRTUMaster_ReadWriteMode.eModbusRTUMaster_ReadRegs THEN 
	fbmodbusmaster.ReadRegs();
		fbmodbusmaster.cbLength := SIZEOF(arrRead);
			fbmodbusmaster.pMemoryAddr := ADR(arrRead); 
END_IF
IF Lynus_Standards.GVL_Bussystems.stDataOfMBRTUMasterKL6xxx[diNrOfMBRTUMasterLine_OUT].eMBRTUReadWriteMode = E_MBRTUMaster_ReadWriteMode.eModbusRTUMaster_WriteMultipleCoils THEN 
	fbmodbusmaster.WriteMultipleCoils();
		fbmodbusmaster.cbLength := SIZEOF(Lynus_Standards.GVL_Bussystems.stDataOfMBRTUMasterKL6xxx[diNrOfMBRTUMasterLine_OUT].arrWriteOutData);
			fbmodbusmaster.pMemoryAddr := ADR(Lynus_Standards.GVL_Bussystems.stDataOfMBRTUMasterKL6xxx[diNrOfMBRTUMasterLine_OUT].arrWriteOutData); 
END_IF
IF Lynus_Standards.GVL_Bussystems.stDataOfMBRTUMasterKL6xxx[diNrOfMBRTUMasterLine_OUT].eMBRTUReadWriteMode = E_MBRTUMaster_ReadWriteMode.eModbusRTUMaster_WriteRegs THEN 
	fbmodbusmaster.WriteRegs(); 
		fbmodbusmaster.cbLength := SIZEOF(Lynus_Standards.GVL_Bussystems.stDataOfMBRTUMasterKL6xxx[diNrOfMBRTUMasterLine_OUT].arrWriteOutData);
			fbmodbusmaster.pMemoryAddr := ADR(Lynus_Standards.GVL_Bussystems.stDataOfMBRTUMasterKL6xxx[diNrOfMBRTUMasterLine_OUT].arrWriteOutData);
END_IF
IF Lynus_Standards.GVL_Bussystems.stDataOfMBRTUMasterKL6xxx[diNrOfMBRTUMasterLine_OUT].eMBRTUReadWriteMode = E_MBRTUMaster_ReadWriteMode.eModbusRTUMaster_WriteSingleCoil THEN 
	fbmodbusmaster.WriteSingleCoil(); 
		fbmodbusmaster.cbLength := SIZEOF(Lynus_Standards.GVL_Bussystems.stDataOfMBRTUMasterKL6xxx[diNrOfMBRTUMasterLine_OUT].arrWriteOutData);
			fbmodbusmaster.pMemoryAddr := ADR(Lynus_Standards.GVL_Bussystems.stDataOfMBRTUMasterKL6xxx[diNrOfMBRTUMasterLine_OUT].arrWriteOutData);
END_IF
IF Lynus_Standards.GVL_Bussystems.stDataOfMBRTUMasterKL6xxx[diNrOfMBRTUMasterLine_OUT].eMBRTUReadWriteMode = E_MBRTUMaster_ReadWriteMode.eModbusRTUMaster_WriteSingleRegister THEN 
	fbmodbusmaster.WriteSingleRegister(); 
		fbmodbusmaster.cbLength := SIZEOF(Lynus_Standards.GVL_Bussystems.stDataOfMBRTUMasterKL6xxx[diNrOfMBRTUMasterLine_OUT].arrWriteOutData);
			fbmodbusmaster.pMemoryAddr := ADR(Lynus_Standards.GVL_Bussystems.stDataOfMBRTUMasterKL6xxx[diNrOfMBRTUMasterLine_OUT].arrWriteOutData);
END_IF

//Order the range of MB Adress when we have a change on that on the slave Functions
IF MEMCMP(ADR(arrMBAdress),ADR(Lynus_Standards.GVL_Bussystems.stDataOfMBRTUMasterKL6xxx[diNrOfMBRTUMasterLine_OUT].arrAllModbusSlaveAdresses),SIZEOF(Lynus_Standards.GVL_Bussystems.stDataOfMBRTUMasterKL6xxx[diNrOfMBRTUMasterLine_OUT].arrAllModbusSlaveAdresses)) <> 0 AND iStateSetMBAdress = 0 THEN
	iStateSetMBAdress := 1;
		bStopReadWrite := TRUE;
			MEMCPY(ADR(arrMBAdress),ADR(Lynus_Standards.GVL_Bussystems.stDataOfMBRTUMasterKL6xxx[diNrOfMBRTUMasterLine_OUT].arrAllModbusSlaveAdresses),SIZEOF(Lynus_Standards.GVL_Bussystems.stDataOfMBRTUMasterKL6xxx[diNrOfMBRTUMasterLine_OUT].arrAllModbusSlaveAdresses));
END_IF

CASE iStateSetMBAdress OF
	
	0://Init
		bStopReadWrite := FALSE;

	1://Set the Actual Adress in use to 0 and Clear old MB Adresses in Array
		bTakeActualAdress := FALSE;
			byActualAdressInUse := 0;
				bySearchMBAdress := 0;
					byPosInArrayMBAdress := 0;	

		FOR byLPMBAdress := 1 TO 247 BY 1 DO
			Lynus_Standards.GVL_Bussystems.stDataOfMBRTUMasterKL6xxx[diNrOfMBRTUMasterLine_OUT].arrAllModbusSlaveAdresses[byLPMBAdress] := 0;
		END_FOR 
			
			iStateSetMBAdress := 2;	
		
	2://Order the new Adresses from lowest to highest
		bySearchMBAdress := bySearchMBAdress + 1;
			bySearchMBAdress := LIMIT(1,bySearchMBAdress,247);			
	
		FOR byLPMBAdress := 1 TO 247 BY 1 DO
			IF arrMBAdress[byLPMBAdress] = bySearchMBAdress THEN
				byPosInArrayMBAdress := byPosInArrayMBAdress + 1;
					byPosInArrayMBAdress := LIMIT(1,byPosInArrayMBAdress,247);
						Lynus_Standards.GVL_Bussystems.stDataOfMBRTUMasterKL6xxx[diNrOfMBRTUMasterLine_OUT].arrAllModbusSlaveAdresses[byPosInArrayMBAdress] := arrMBAdress[byLPMBAdress]; 	
			END_IF
		END_FOR  
		
		//Done
		IF bySearchMBAdress >= 247 THEN 
			iStateSetMBAdress := 0;
				MEMCPY(ADR(arrMBAdress),ADR(Lynus_Standards.GVL_Bussystems.stDataOfMBRTUMasterKL6xxx[diNrOfMBRTUMasterLine_OUT].arrAllModbusSlaveAdresses),SIZEOF(Lynus_Standards.GVL_Bussystems.stDataOfMBRTUMasterKL6xxx[diNrOfMBRTUMasterLine_OUT].arrAllModbusSlaveAdresses));
		END_IF 
	
END_CASE

//Check the Modbus Adresses from each Slave Device
FPProcessCompleted(CLK:= Lynus_Standards.GVL_Bussystems.stDataOfMBRTUMasterKL6xxx[diNrOfMBRTUMasterLine_OUT].bReadWriteIsDone, Q=> );
	FPError(CLK:= fbmodbusmaster.Error, Q=> );

bySmallestAdress := 247;	
	FOR byLPSmallestAdress := 1 TO 247 BY 1 DO
		IF Lynus_Standards.GVL_Bussystems.stDataOfMBRTUMasterKL6xxx[diNrOfMBRTUMasterLine_OUT].arrAllModbusSlaveAdresses[byLPSmallestAdress] < bySmallestAdress AND Lynus_Standards.GVL_Bussystems.stDataOfMBRTUMasterKL6xxx[diNrOfMBRTUMasterLine_OUT].arrAllModbusSlaveAdresses[byLPSmallestAdress] <> 0 THEN bySmallestAdress := Lynus_Standards.GVL_Bussystems.stDataOfMBRTUMasterKL6xxx[diNrOfMBRTUMasterLine_OUT].arrAllModbusSlaveAdresses[byLPSmallestAdress]; END_IF
	END_FOR
byBiggestAdress := 0;
	FOR byLPBiggestAdress := 1 TO 247 BY 1 DO
		IF Lynus_Standards.GVL_Bussystems.stDataOfMBRTUMasterKL6xxx[diNrOfMBRTUMasterLine_OUT].arrAllModbusSlaveAdresses[byLPBiggestAdress] > byBiggestAdress THEN byBiggestAdress := Lynus_Standards.GVL_Bussystems.stDataOfMBRTUMasterKL6xxx[diNrOfMBRTUMasterLine_OUT].arrAllModbusSlaveAdresses[byLPBiggestAdress]; END_IF  
	END_FOR
//Take the Next Adress after the Read/write is done
IF FPProcessCompleted.Q OR FPError.Q THEN
	bTakeActualAdress := TRUE;
		FOR byLPActualAdress := 1 TO 247 BY 1 DO
			IF Lynus_Standards.GVL_Bussystems.stDataOfMBRTUMasterKL6xxx[diNrOfMBRTUMasterLine_OUT].arrAllModbusSlaveAdresses[byLPActualAdress] > byActualAdressInUse THEN 
				byActualAdressInUse := Lynus_Standards.GVL_Bussystems.stDataOfMBRTUMasterKL6xxx[diNrOfMBRTUMasterLine_OUT].arrAllModbusSlaveAdresses[byLPActualAdress]; 
					EXIT;
			END_IF
		END_FOR		
END_IF

//Count the Number of RTU Slaves
byNumberOfTotalSlaves := 0;
	FOR byLPNumbersOfTotalSlaves := 1 TO 247 BY 1 DO
		IF Lynus_Standards.GVL_Bussystems.stDataOfMBRTUMasterKL6xxx[diNrOfMBRTUMasterLine_OUT].arrAllModbusSlaveAdresses[byLPNumbersOfTotalSlaves] <> 0 THEN byNumberOfTotalSlaves := byNumberOfTotalSlaves + 1; END_IF
	END_FOR

FNInitSmall(CLK:= bySmallestAdress = 247, Q=> );

IF byActualAdressInUse <> byActualAdressInUse_CP THEN bAdressHasChanged := TRUE; byActualAdressInUse_CP := byActualAdressInUse; ELSE bAdressHasChanged := FALSE; END_IF 

IF ((FPError.Q OR FPProcessCompleted.Q) AND NOT bAdressHasChanged) OR FNInitSmall.Q OR bySmallestAdress = byBiggestAdress THEN byActualAdressInUse := bySmallestAdress; END_IF

timTimout(IN:= Lynus_Standards.GVL_Bussystems.stDataOfMBRTUMasterKL6xxx[diNrOfMBRTUMasterLine_OUT].bReadWriteIsDone, PT:= , Q=> , ET=> );

IF FPProcessCompleted.Q OR timTimout.Q THEN Lynus_Standards.GVL_Bussystems.stDataOfMBRTUMasterKL6xxx[diNrOfMBRTUMasterLine_OUT].bReadWriteIsDone := FALSE; END_IF

IF NOT bTakeActualAdress THEN 
	fbmodbusmaster.UnitID := bySmallestAdress;
ELSE
	fbmodbusmaster.UnitID := byActualAdressInUse;
END_IF

fbmodbusmaster(
	UnitID:= , 
	Quantity:= Lynus_Standards.GVL_Bussystems.stDataOfMBRTUMasterKL6xxx[diNrOfMBRTUMasterLine_OUT].wNumberOfRegister, 
	MBAddr:= Lynus_Standards.GVL_Bussystems.stDataOfMBRTUMasterKL6xxx[diNrOfMBRTUMasterLine_OUT].wModbusRegister, 
	cbLength:= , 
	pMemoryAddr:= , 
	Execute:= Lynus_Standards.GVL_Bussystems.stDataOfMBRTUMasterKL6xxx[diNrOfMBRTUMasterLine_OUT].bSlaveStartReadOrWrite AND bTerminalIsConfigured AND NOT timDissableFunctions.Q AND NOT bStopReadWrite, 
	Timeout:= , 
	BUSY=> , 
	Error=> , 
	ErrorId=> , 
	cbRead=> );	
	
(*------------------------------------------------------------------Busy Flag----------------------------------------------------------------------------*)

IF NOT bTerminalIsConfigured THEN
	bBusy := fbKL6xxxConfig.Busy;
ELSE
	bBusy := fbmodbusmaster.BUSY;
END_IF

//When we have a change on the MB Adress List we set the Function always on Busy that al other Slave Functions Stops in the Init Step
IF bStopReadWrite THEN bBusy := TRUE; END_IF

FNBusy(CLK:= fbmodbusmaster.BUSY, Q=> );

(*------------------------------------------------------------------Error and Warning----------------------------------------------------------------------------*)

IF timDissableFunctions.Q THEN fbModbusRTUMessage.bWarning := TRUE; fbModbusRTUMessage.iWarningCode := 0; ELSE fbModbusRTUMessage.bWarning := FALSE; END_IF   
	IF (Lynus_Standards.GVL_Bussystems.diNumberOfMBRTUMasters > Constants_Bussystems.diMaxNumberOfMBRTUMasterKL6xxx) OR (NOT bTerminalIsConfigured AND fbKL6xxxConfig.Error) OR (bTerminalIsConfigured AND fbmodbusmaster.Error) OR bStopReadWrite THEN 
		fbModbusRTUMessage.bError := TRUE;
	ELSE
		fbModbusRTUMessage.bError := FALSE;
	END_IF

IF Lynus_Standards.GVL_Bussystems.diNumberOfMBRTUMasters > Constants_Bussystems.diMaxNumberOfMBRTUMasterKL6xxx THEN
	fbModbusRTUMessage.iErrorCode := 1;	
ELSIF NOT bTerminalIsConfigured THEN 
	IF fbKL6xxxConfig.Error THEN 
		fbModbusRTUMessage.iErrorCode := 2; 
	END_IF
//When we have a change on the MB Adress List we set the Function always on Error that al other Slave Functions go back to the Init Step
ELSIF bStopReadWrite THEN
	fbModbusRTUMessage.iErrorCode := 2; 
ELSE
	IF fbmodbusmaster.ErrorId = 1 THEN fbModbusRTUMessage.iErrorCode := 3; END_IF
	IF fbmodbusmaster.ErrorId = 2 THEN fbModbusRTUMessage.iErrorCode := 4; END_IF
	IF fbmodbusmaster.ErrorId = 3 THEN fbModbusRTUMessage.iErrorCode := 5; END_IF
	IF fbmodbusmaster.ErrorId = 4 THEN fbModbusRTUMessage.iErrorCode := 6; END_IF
	IF fbmodbusmaster.ErrorId = 5 THEN fbModbusRTUMessage.iErrorCode := 7; END_IF
	IF fbmodbusmaster.ErrorId = 6 THEN fbModbusRTUMessage.iErrorCode := 8; END_IF
	IF fbmodbusmaster.ErrorId = 7 THEN fbModbusRTUMessage.iErrorCode := 9; END_IF
	IF fbmodbusmaster.ErrorId = 8 THEN fbModbusRTUMessage.iErrorCode := 10; END_IF
	IF fbmodbusmaster.ErrorId = 16#A THEN fbModbusRTUMessage.iErrorCode := 11; END_IF
	IF fbmodbusmaster.ErrorId = 16#B THEN fbModbusRTUMessage.iErrorCode := 12; END_IF
	IF fbmodbusmaster.ErrorId = 16#20 THEN fbModbusRTUMessage.iErrorCode := 13; END_IF
	IF fbmodbusmaster.ErrorId = 16#21 THEN fbModbusRTUMessage.iErrorCode := 14; END_IF
	IF fbmodbusmaster.ErrorId = 16#22 THEN fbModbusRTUMessage.iErrorCode := 15; END_IF
	IF fbmodbusmaster.ErrorId = 16#23 THEN fbModbusRTUMessage.iErrorCode := 16; END_IF
	IF fbmodbusmaster.ErrorId = 16#24 THEN fbModbusRTUMessage.iErrorCode := 17; END_IF
	IF fbmodbusmaster.ErrorId = 16#25 THEN fbModbusRTUMessage.iErrorCode := 18; END_IF
	IF fbmodbusmaster.ErrorId = 102 THEN fbModbusRTUMessage.iErrorCode := 19; END_IF
	IF fbmodbusmaster.ErrorId = 103 THEN fbModbusRTUMessage.iErrorCode := 20; END_IF
	IF fbmodbusmaster.ErrorId = 107 THEN fbModbusRTUMessage.iErrorCode := 21; END_IF
	IF fbmodbusmaster.ErrorId = 110 THEN fbModbusRTUMessage.iErrorCode := 22; END_IF
	IF fbmodbusmaster.ErrorId = 120 THEN fbModbusRTUMessage.iErrorCode := 23; END_IF
	IF fbmodbusmaster.ErrorId = 150 THEN fbModbusRTUMessage.iErrorCode := 24; END_IF
	IF fbmodbusmaster.ErrorId = 232 THEN fbModbusRTUMessage.iErrorCode := 25; END_IF
	IF fbmodbusmaster.ErrorId = 233 THEN fbModbusRTUMessage.iErrorCode := 26; END_IF
END_IF

fbModbusRTUMessage(
	bTerminalConfigured:= bTerminalIsConfigured, 
	bError:= , 
	bWarning:= , 
	iWarningCode:= , 
	iErrorCode:= , 
	byErrorWarning=> byErrorWarning, 
	eMessageMBRTUMaster=> eMessageMBRTUMaster);

//Set this Flag after a Error and Reset after next Read or Write command without Error	
IF FPError.Q THEN bErrorIsActive := TRUE; END_IF
	IF FNBusy.Q AND NOT fbmodbusmaster.Error THEN bErrorIsActive := FALSE; END_IF	
	
FPErrorIsActive(CLK:= bErrorIsActive, Q=> );
	
(*-----------------------------------------------------------Handle data to Global structure for Modbus RTU Communication-----------------------------------------------------------------*)

CASE iStateGVLData OF
	
	0://Init Step
		byWaitInStep := 0;
			diCounterForGVL := 1;
	
	1://Wait for 4 Steps before clean al Data on GVL
		byWaitInStep := byWaitInStep + 1;
			IF byWaitInStep >= 4 AND fbNumberDevice.bNumberIsCalculatet THEN iStateGVLData := 2; END_IF
				//To much Devices, back to the Init step
				IF byWaitInStep >= 4 AND NOT fbNumberDevice.bNumberIsCalculatet THEN iStateGVLData := 0; END_IF	
			
	2://Clear all Data in GVL
	//Some Parts in the GVL Reset the Slave. Otherwise there will be problems when writing the new addresses to the array in the GVL.
	Lynus_Standards.GVL_Bussystems.stDataOfMBRTUMasterKL6xxx[diCounterForGVL].bMasterIsBusy := FALSE;	
		Lynus_Standards.GVL_Bussystems.stDataOfMBRTUMasterKL6xxx[diCounterForGVL].bTerminalIsConfigured := FALSE;	
			Lynus_Standards.GVL_Bussystems.stDataOfMBRTUMasterKL6xxx[diCounterForGVL].byNumberOfSlaves := 0;
				Lynus_Standards.GVL_Bussystems.stDataOfMBRTUMasterKL6xxx[diCounterForGVL].byErrorWarning := 0;
					Lynus_Standards.GVL_Bussystems.stDataOfMBRTUMasterKL6xxx[diCounterForGVL].byActualMBAdressInProgrss := 0;
						Lynus_Standards.GVL_Bussystems.stDataOfMBRTUMasterKL6xxx[diCounterForGVL].bNoNewMBusAdress := FALSE;	
														 		
		diCounterForGVL := diCounterForGVL + 1;
			diCounterForGVL := LIMIT(0,diCounterForGVL,Constants_Bussystems.diMaxNumberOfMBRTUMasterKL6xxx);
				//Back to the init step
				IF diCounterForGVL >= Constants_Bussystems.diMaxNumberOfMBRTUMasterKL6xxx THEN iStateGVLData := 0; END_IF

END_CASE 
	
IF diNrOfMBRTUMasterLine_OUT > 0 AND fbNumberDevice.bNumberIsCalculatet THEN  
	Lynus_Standards.GVL_Bussystems.stDataOfMBRTUMasterKL6xxx[diNrOfMBRTUMasterLine_OUT].bMasterIsBusy := bBusy;
		Lynus_Standards.GVL_Bussystems.stDataOfMBRTUMasterKL6xxx[diNrOfMBRTUMasterLine_OUT].byErrorWarning := byErrorWarning;
			Lynus_Standards.GVL_Bussystems.stDataOfMBRTUMasterKL6xxx[diNrOfMBRTUMasterLine_OUT].bTerminalIsConfigured := bTerminalIsConfigured;
				Lynus_Standards.GVL_Bussystems.stDataOfMBRTUMasterKL6xxx[diNrOfMBRTUMasterLine_OUT].byActualMBAdressInProgrss := fbmodbusmaster.UnitID;
					Lynus_Standards.GVL_Bussystems.stDataOfMBRTUMasterKL6xxx[diNrOfMBRTUMasterLine_OUT].byNumberOfSlaves := byNumberOfTotalSlaves;
						Lynus_Standards.GVL_Bussystems.stDataOfMBRTUMasterKL6xxx[diCounterForGVL].bNoNewMBusAdress := bStopReadWrite;
						IF FNBusy.Q THEN
							IF NOT fbmodbusmaster.Error THEN
								Lynus_Standards.GVL_Bussystems.stDataOfMBRTUMasterKL6xxx[diNrOfMBRTUMasterLine_OUT].arrReadOutData := arrRead;
							ELSE
								//Workarround about internal Beckhoff Lib Error 
								IF FPErrorIsActive.Q THEN 
									MEMCPY(ADR(fbmodbusmaster),ADR(fbmodbusmaster_Init),SIZEOF(fbmodbusmaster_Init));
								END_IF
							END_IF
						END_IF	
END_IF	
	
(*----------------------------------------------------------Save persistent data----------------------------------------------------------------*)

arrPD[1](lrValue:= BOOL_TO_LREAL(bTerminalIsConfigured), bEventBasedActive=> );
arrPD[2](lrValue:= INT_TO_LREAL(eDeviceType), bEventBasedActive=> );

END_FUNCTION_BLOCK

// ---- FB/FB_Shelly_HT_Helper.TcPOU
FUNCTION_BLOCK FB_Shelly_HT_Helper
VAR_INPUT
	bSend				: BOOL;
END_VAR

VAR_IN_OUT
	fbClient			: FB_IotHttpClient;
END_VAR

VAR_OUTPUT
	bBusy				: BOOL;
	bError				: BOOL;
	lr_Temperature		: LREAL;						//Received Value
	lr_Humidity			: LREAL;
END_VAR

VAR
	fbRequestStatus		: FB_IotHttpRequest;
	fbJson				: FB_JsonDomParser;
	nState				: UDINT;
	RisingEdge			: R_TRIG;
	timTimeout			: TON;
	tTimeOut			: TIME := T#50S;
	bGetContentResult	: BOOL;
	sContentStatus		: STRING(511);
	sContentM0			: STRING(511);
	sContentM1			: STRING(511);
	sContentM2			: STRING(511);
	
	bGetJsonResult		: BOOL;
	jsonDoc				: SJsonValue;
	jsonVal				: SJsonValue;
	
	nReqCount			: UDINT;	
	nResCount			: UDINT;
	nValidResCount		: UDINT;
	nErrCount			: UDINT;
	x: INT;
END_VAR

//Timer for Timeout
timTimeout(IN:= nState = 1 AND bBusy, PT:= tTimeOut, Q=> , ET=> );
	IF timTimeout.Q THEN 
		nState := 0;
		bBusy := FALSE;
	END_IF

RisingEdge(CLK:= bSend );
CASE nState OF
0:	
	IF RisingEdge.Q THEN 
		IF 
			fbRequestStatus.SendRequest(sUri:='/status', fbClient:=fbClient, eRequestType:=ETcIotHttpRequestType.HTTP_Get, 0, 0, 0) THEN				
			nState:= 1;
			nReqCount:= nReqCount+1;
			bBusy:= TRUE;
			bError:= FALSE;
		END_IF					
	END_IF
1:
	x:=x+1;
	IF  NOT fbRequestStatus.bBusy THEN
		bError:= TRUE;
			
		IF NOT fbRequestStatus.bError THEN				 
			bGetContentResult:= fbRequestStatus.GetContent(pContent:= ADR(sContentStatus), nContentSize:= SIZEOF(sContentStatus), bSetNullTermination:= TRUE);
			IF fbRequestStatus.nStatusCode >= 200 AND fbRequestStatus.nStatusCode < 300 THEN
				bGetJsonResult:= FALSE;
				jsonDoc:= fbRequestStatus.GetJsonDomContent(fbJson);
				IF jsonDoc <> 0 THEN
					bGetJsonResult:= TRUE;
					IF fbJson.HasMember(jsonDoc, 'tmp.value')  THEN
						jsonVal:= fbJson.FindMember(jsonDoc, 'tmp.value');
						nValidResCount:= nValidResCount+1;
						IF fbJson.IsDouble(jsonVal) THEN							
							lr_Temperature:= fbJson.GetDouble(jsonVal);									
						END_IF
						bError:= FALSE;
					END_IF
					IF fbJson.HasMember(jsonDoc, 'hum.value')  THEN
						jsonVal:= fbJson.FindMember(jsonDoc, 'hum.value');
						nValidResCount:= nValidResCount+1;
						IF fbJson.IsDouble(jsonVal) THEN							
							lr_Humidity:= fbJson.GetDouble(jsonVal);									
						END_IF
						bError:= FALSE;
					END_IF
				END_IF		
				nResCount:= nResCount+1;			
			END_IF
		END_IF
		
		nState:= 0;
		bBusy:= FALSE;
		IF bError THEN
			nErrCount:= nErrCount+1;
		END_IF
	END_IF  	
END_CASE

END_FUNCTION_BLOCK

// ---- POUs/MAIN.TcPOU
PROGRAM MAIN
VAR
END_VAR

(* Hallo Git *)

END_PROGRAM

// ---- POUs/prgEM.TcPOU
PROGRAM prgEM
VAR
		// Grid Objekt H 3-phase, 400V
	fb_UV_Garderobe					: FB_Shelly_3EM;
	
	lrPower_UV_Garderobe_TotalkW		: LREAL;			//{#lynus.ag#()}
	lrEnergy_UV_Garderobe_Total			: LREAL;			//{#lynus.ag#()}
	lrCurrent_UV_Garderobe_L1			: LREAL;			//{#lynus.ag#()}
	lrCurrent_UV_Garderobe_L2			: LREAL;			//{#lynus.ag#()}
	lrCurrent_UV_Garderobe_L3			: LREAL;			//{#lynus.ag#()}
	lrVoltage_UV_Garderobe_L1			: LREAL;			//{#lynus.ag#()}
	lrVoltage_UV_Garderobe_L2			: LREAL;			//{#lynus.ag#()}
	lrVoltage_UV_Garderobe_L3			: LREAL;			//{#lynus.ag#()}


	fb_Temperature_1				: FB_Shelly_hT;
	fb_Temperature_2				: FB_Shelly_HTplus;

	str_ip: STRING(15):='172.32.12.127';
	m_Start1: BOOL;
	m_Start2: BOOL;
	lrTemp1: LREAL;
	lrTemp2: LREAL;
END_VAR

	// Grid Objekt H 3-phase, 400V
fb_UV_Garderobe(
	bStart:= , 
	tDelayRequest:= T#20S, 
	sHostname:= '172.32.12.121', 
	bValidResult=> , 
	bBusy=> , 
	bError=> , 
	bDone=> , 
	hrErrorCode=> ,
	lrtotalpower=> ,
	lrpowerL1=> ,
	lrpowerL2=> ,
	lrpowerL3=> ,
	lrcurrentL1=> lrCurrent_UV_Garderobe_L1,
	lrcurrentL2=> lrCurrent_UV_Garderobe_L2,
	lrcurrentL3=> lrCurrent_UV_Garderobe_L3,
	lrvoltageL1=> lrVoltage_UV_Garderobe_L1,
	lrvoltageL2=> lrVoltage_UV_Garderobe_L2,
	lrvoltageL3=> lrVoltage_UV_Garderobe_L3,
	lrenergyL1=> ,
	lrenergyL2=> ,
	lrenergyL3=>  );

lrPower_UV_Garderobe_TotalkW := 	fb_UV_Garderobe.lrtotalpower / 1000;
// sum-up energy
lrEnergy_UV_Garderobe_Total :=  fb_UV_Garderobe.lrenergyL1 + fb_UV_Garderobe.lrenergyL2 + fb_UV_Garderobe.lrenergyL3;


fb_Temperature_1(
	bStart:= m_Start1, 
	tDelayRequest:= T#10S, 
	sHostname:= '172.32.12.127', 
	bValidResult=> , 
	bBusy=> , 
	bError=> , 
	bDone=> , 
	bConnected=> , 
	lr_Temperature=> , 
	lr_Humidity=> , 
	hrErrorCode=> );
	


fb_Temperature_2(
	bStart:= m_Start2, 
	tDelayRequest:= T#10S, 
	sHostname:= '172.32.12.124', 
	bValidResult=> , 
	bBusy=> , 
	bError=> , 
	bDone=> , 
	bConnected=> , 
	lr_Temperature=> , 
	lr_Humidity=> , 
	hrErrorCode=> );
	
IF fb_Temperature_1.lr_Temperature <> 0  THEN 
	lrTemp1 :=  fb_Temperature_1.lr_Temperature;
END_IF
IF fb_Temperature_2.lr_Temperature<>0 THEN
	lrTemp2 :=  fb_Temperature_2.lr_Temperature;
END_IF

END_PROGRAM
